FUNCTION Buffer_Layout_Set_Int_Array : UINT
VAR_INPUT
END_VAR
VAR
END_VAR

END_FUNCTION

(* stored: Version 1.1.0.1, ProductVersion 3.1.4024.10
   POU Buffer_Layout_Set_Int_Array: Id {add70a58-5de9-4c97-bed6-2b6c490363be}, SpecialFunc None *)
